(* CODESYS project PLS2 Trykkregulering 19.07.2021.export

Project tree, tasks and I/O mapping:
  application PLS2_Trykkregulering
    task PLC_Task (cyclic, interval 100 ms, priority 10, watchdog 90 ms x 1) calls PLC_PRG
    task TrendRecordingTask (cyclic, interval 100 ms, priority 15) calls VisuTrendStorageAccess.GlobalInstances.g_TrendRecordingManager.CyclicCall
    task VISU_TASK (cyclic, interval 100 ms, priority 15) calls VisuElems.Visu_Prg
    GlobalData/
      global variables HMI
      global variables IO
      global variables Local
      global variables SIM
      global variables STATUS
    program Alarms [ST]
    program Control [ST]
    program Initialize [ST]
    program Inputs [ST]
    program Outputs [ST]
    program PLC_PRG [ST]
    function RestartOpcUaMqttLinkOnDownload [ST]
    function RestartOpcUaMqttLinkOnOnlineChange [ST]
    program Simulation [ST]
    global variables PersistentVars
    visualisation Visualization
*)

// PLS2_Trykkregulering/PersistentVars
{attribute 'qualified_only'}
VAR_GLOBAL PERSISTENT RETAIN
	// Generated instance path of persistent variable
	HMI.AliveCounterPlc2Pv: AliveHmiPv;
	// Generated instance path of persistent variable
	HMI.DeliveryPump1Cmd: ControlAnalogHmiCmd;
	// Generated instance path of persistent variable
	HMI.DeliveryPump1Pv: ControlAnalogHmiPv;
	// Generated instance path of persistent variable
	HMI.DeliveryPump2Cmd: ControlAnalogHmiCmd;
	// Generated instance path of persistent variable
	HMI.DeliveryPump2Pv: ControlAnalogHmiPv;
	// Generated instance path of persistent variable
	HMI.DeliveryPump3Cmd: ControlAnalogHmiCmd;
	// Generated instance path of persistent variable
	HMI.DeliveryPump3Pv: ControlAnalogHmiPv;
	// Generated instance path of persistent variable
	HMI.DeliveryPumpPIDCmd: PIDHmiCmd;
	// Generated instance path of persistent variable
	HMI.DeliveryPumpPIDPv: PIDHmiPv;
	// Generated instance path of persistent variable
	HMI.DeliveryPumpWorkDistPv: WorkDistributorHmiPv;
	// Generated instance path of persistent variable
	HMI.TreatmentPressureCmd: SignalAnalogHmiCmd;
	// Generated instance path of persistent variable
	HMI.TreatmentPressurePv: SignalAnalogHmiPv;
	// Generated instance path of persistent variable
	HMI.ConsumerPressureCmd: SignalAnalogHmiCmd;
	// Generated instance path of persistent variable
	HMI.ConsumerPressurePv: SignalAnalogHmiPv;
END_VAR

// PLS2_Trykkregulering/GlobalData/HMI
{attribute 'qualified_only'}
VAR_GLOBAL PERSISTENT RETAIN
AliveCounterPlc2Pv:AliveHmiPv;

DeliveryPump1Cmd:ControlAnalogHmiCmd;
DeliveryPump1Pv:ControlAnalogHmiPv;
DeliveryPump2Cmd:ControlAnalogHmiCmd;
DeliveryPump2Pv:ControlAnalogHmiPv;
DeliveryPump3Cmd:ControlAnalogHmiCmd;
DeliveryPump3Pv:ControlAnalogHmiPv;
DeliveryPumpPIDCmd:PIDHmiCmd;
DeliveryPumpPIDPv:PIDHmiPv;
DeliveryPumpWorkDistPv:WorkDistributorHmiPv;
TreatmentPressureCmd:SignalAnalogHmiCmd;
TreatmentPressurePv:SignalAnalogHmiPv;
ConsumerPressureCmd:SignalAnalogHmiCmd;
ConsumerPressurePv:SignalAnalogHmiPv;
END_VAR

// PLS2_Trykkregulering/GlobalData/IO
{attribute 'qualified_only'}
VAR_GLOBAL
AI_DeliveryPump1SpeedPv:REAL;
AI_DeliveryPump2SpeedPv:Real;
AI_DeliveryPump3SpeedPv:Real;

AO_DeliveryPump1ControlValue:real;
AO_DeliveryPump2ControlValue:real;
AO_DeliveryPump3ControlValue:REAL;

AI_ConsumerPressurePv:REAL;
AI_TreatmentPressurePv:REAL;
END_VAR

// PLS2_Trykkregulering/GlobalData/Local
{attribute 'qualified_only'}
VAR_GLOBAL
DeliveryPump1:ControlAnalogFB;
DeliveryPump2:ControlAnalogFB;
DeliveryPump3:ControlAnalogFB;
DeliveryPumpPID:PIDFB;
DeliveryPumpWorkDist:WorkDistributorFB;
TreatmentPressure:SignalAnalogFB;
ConsumerPressure:SignalAnalogFB;
END_VAR

// PLS2_Trykkregulering/GlobalData/SIM
{attribute 'qualified_only'}
VAR_GLOBAL
	Disturbance:REAL;
	Process_y:REAL;
	Process:REAL;
	Ref:REAL;
	Output:REAL;
END_VAR

// PLS2_Trykkregulering/GlobalData/STATUS
{attribute 'qualified_only'}
VAR_GLOBAL
	OpcUaMqttLinkStatus: OpcUa_Mqtt_Status;
END_VAR

// PLS2_Trykkregulering/PLC_PRG
PROGRAM PLC_PRG
VAR
	_firstScan:BOOL := TRUE;
	_counter:INT;
	_lastRun:STRING;
END_VAR



// Signaling that the PLC is alive
Hmi.AliveCounterPlc2Pv._tagId := 'AliveCounterPlc2Pv';
Hmi.AliveCounterPlc2Pv._type := 'AliveHmi';
Hmi.AliveCounterPlc2Pv._owner := 'plc2';
HMI.AliveCounterPlc2Pv.CounterPv := HMI.AliveCounterPlc2Pv.CounterPv + 1;

_counter := STATUS.OpcUaMqttLinkStatus.AliveCounterPv;
_lastRun := STATUS.OpcUaMqttLinkStatus.LastRun;

IF _firstScan THEN
	Initialize();
END_IF
Inputs();
Alarms();
Control();
Outputs();
Simulation();





// Always last
_firstScan := FALSE;

END_PROGRAM

// PLS2_Trykkregulering/Initialize
PROGRAM Initialize
VAR
END_VAR



Hmi.DeliveryPumpPIDCmd.Tag := 'PID01';
Hmi.DeliveryPumpPIDCmd.Description := 'Regulator for controling pressure';
Hmi.DeliveryPumpPIDCmd.Auto := TRUE;
Hmi.DeliveryPumpPIDCmd.EnableK := TRUE;
Hmi.DeliveryPumpPIDCmd.EnableI := TRUE;
Hmi.DeliveryPumpPIDCmd.EnableD := TRUE;
Hmi.DeliveryPumpPIDCmd.K := 8.0;
Hmi.DeliveryPumpPIDCmd.Ti := 5.5;
Hmi.DeliveryPumpPIDCmd.Td := 0.5;
Hmi.DeliveryPumpPIDCmd.N := 10.0;
Hmi.DeliveryPumpPIDCmd.TrackingGain := 1.0;
Hmi.DeliveryPumpPIDCmd.u0 := 50.0;


HMI.DeliveryPump1Cmd.Tag := 'P01';
HMI.DeliveryPump1Cmd.Description := 'Delivery pump 1';
HMI.DeliveryPump1Cmd.Auto := TRUE;
HMI.DeliveryPump1Cmd.ManualControlValue_Cmd := 50.0;
HMI.DeliveryPump1Cmd.AlarmControlFailedLimit := 10.0;
HMI.DeliveryPump1Cmd.AlarmControlFailed.Description := 'Failed to control Delivery Pump 1';
HMI.DeliveryPump1Cmd.AlarmControlFailed.Delay.OnDelayLimit := 10.0;
HMI.DeliveryPump1Cmd.AlarmControlFailed.Delay.OffDelayLimit := 10.0;
HMI.DeliveryPump1Cmd.AlarmControlFailed.Acknowledged := TRUE;

HMI.DeliveryPump2Cmd.Tag := 'P02';
HMI.DeliveryPump2Cmd.Description := 'Delivery pump 2';
HMI.DeliveryPump2Cmd.Auto := TRUE;
HMI.DeliveryPump2Cmd.ManualControlValue_Cmd := 50.0;
HMI.DeliveryPump2Cmd.AlarmControlFailedLimit := 10.0;
HMI.DeliveryPump2Cmd.AlarmControlFailed.Description := 'Failed to control Delivery Pump 2';
HMI.DeliveryPump2Cmd.AlarmControlFailed.Delay.OnDelayLimit := 10.0;
HMI.DeliveryPump2Cmd.AlarmControlFailed.Delay.OffDelayLimit := 10.0;
HMI.DeliveryPump2Cmd.AlarmControlFailed.Acknowledged := TRUE;

HMI.DeliveryPump3Cmd.Tag := 'P03';
HMI.DeliveryPump3Cmd.Description := 'Delivery pump 2';
HMI.DeliveryPump3Cmd.Auto := TRUE;
HMI.DeliveryPump3Cmd.ManualControlValue_Cmd := 50.0;
HMI.DeliveryPump3Cmd.AlarmControlFailedLimit := 10.0;
HMI.DeliveryPump3Cmd.AlarmControlFailed.Description := 'Failed to control Delivery Pump 3';
HMI.DeliveryPump3Cmd.AlarmControlFailed.Delay.OnDelayLimit := 10.0;
HMI.DeliveryPump3Cmd.AlarmControlFailed.Delay.OffDelayLimit := 10.0;
HMI.DeliveryPump3Cmd.AlarmControlFailed.Acknowledged := TRUE;

Hmi.TreatmentPressureCmd.Tag := 'PT02';
Hmi.TreatmentPressureCmd.Description := 'Treatment pressure';
Hmi.TreatmentPressureCmd.AlarmHysteresis := 3.0;
Hmi.TreatmentPressureCmd.AlarmHighHighLimit := 90.0;
Hmi.TreatmentPressureCmd.AlarmHighLimit := 80.0;
Hmi.TreatmentPressureCmd.AlarmLowLowLimit := 10.0;
Hmi.TreatmentPressureCmd.AlarmLowLimit := 20.0;
Hmi.TreatmentPressureCmd.AlarmHigh.Description := 'High Treatment Pressure';
Hmi.TreatmentPressureCmd.AlarmHighHigh.Description := 'High high Treatment Pressure';
Hmi.TreatmentPressureCmd.AlarmLow.Description := 'Low Treatment Pressure';
Hmi.TreatmentPressureCmd.AlarmLowLow.Description := 'Low low Treatment Pressure';
Hmi.TreatmentPressureCmd.AlarmHigh.Delay.OnDelayLimit := 1.0;
Hmi.TreatmentPressureCmd.AlarmHigh.Delay.OffDelayLimit := 1.0;
Hmi.TreatmentPressureCmd.AlarmHighHigh.Delay.OnDelayLimit := 1.0;
Hmi.TreatmentPressureCmd.AlarmHighHigh.Delay.OffDelayLimit := 1.0;
Hmi.TreatmentPressureCmd.AlarmLow.Delay.OnDelayLimit := 1.0;
Hmi.TreatmentPressureCmd.AlarmLow.Delay.OffDelayLimit := 1.0;
Hmi.TreatmentPressureCmd.AlarmLowLow.Delay.OnDelayLimit := 1.0;
Hmi.TreatmentPressureCmd.AlarmLowLow.Delay.OffDelayLimit := 1.0;
Hmi.TreatmentPressureCmd.InputScaling.InputUnit := 'na';
Hmi.TreatmentPressureCmd.InputScaling.OutputUnit := 'bar';
Hmi.TreatmentPressureCmd.InputScaling.InputMax_Cmd := 100.0;
Hmi.TreatmentPressureCmd.InputScaling.InputMin_Cmd := 0.0;
Hmi.TreatmentPressureCmd.InputScaling.OutputMax_Cmd := 100.0;
Hmi.TreatmentPressureCmd.InputScaling.OutputMin_Cmd := 0.0;

Hmi.ConsumerPressureCmd.Tag := 'PT03';
Hmi.ConsumerPressureCmd.Description := 'Consumer pressure';
Hmi.ConsumerPressureCmd.AlarmHysteresis := 3.0;
Hmi.ConsumerPressureCmd.AlarmHighHighLimit := 90.0;
Hmi.ConsumerPressureCmd.AlarmHighLimit := 80.0;
Hmi.ConsumerPressureCmd.AlarmLowLowLimit := 10.0;
Hmi.ConsumerPressureCmd.AlarmLowLimit := 20.0;
Hmi.ConsumerPressureCmd.AlarmHigh.Description := 'High Consumer Pressure';
Hmi.ConsumerPressureCmd.AlarmHighHigh.Description := 'High high Consumer Pressure';
Hmi.ConsumerPressureCmd.AlarmLow.Description := 'Low Consumer Pressure';
Hmi.ConsumerPressureCmd.AlarmLowLow.Description := 'Low low Consumer Pressure';
Hmi.ConsumerPressureCmd.AlarmHigh.Delay.OnDelayLimit := 1.0;
Hmi.ConsumerPressureCmd.AlarmHigh.Delay.OffDelayLimit := 1.0;
Hmi.ConsumerPressureCmd.AlarmHighHigh.Delay.OnDelayLimit := 1.0;
Hmi.ConsumerPressureCmd.AlarmHighHigh.Delay.OffDelayLimit := 1.0;
Hmi.ConsumerPressureCmd.AlarmLow.Delay.OnDelayLimit := 1.0;
Hmi.ConsumerPressureCmd.AlarmLow.Delay.OffDelayLimit := 1.0;
Hmi.ConsumerPressureCmd.AlarmLowLow.Delay.OnDelayLimit := 1.0;
Hmi.ConsumerPressureCmd.AlarmLowLow.Delay.OffDelayLimit := 1.0;
Hmi.ConsumerPressureCmd.InputScaling.InputUnit := 'na';
Hmi.ConsumerPressureCmd.InputScaling.OutputUnit := 'bar';
Hmi.ConsumerPressureCmd.InputScaling.InputMax_Cmd := 100.0;
Hmi.ConsumerPressureCmd.InputScaling.InputMin_Cmd := 0.0;
Hmi.ConsumerPressureCmd.InputScaling.OutputMax_Cmd := 100.0;
Hmi.ConsumerPressureCmd.InputScaling.OutputMin_Cmd := 0.0;

END_PROGRAM

// PLS2_Trykkregulering/Control
PROGRAM Control
VAR
	
END_VAR



// Regulator block
Local.DeliveryPumpPID(_id := 'DeliveryPumpPID', _owner := 'plc2',
	InputReference := 6.0,
	ProcessMeasure := IO.AI_ConsumerPressurePv,
	Ts := 0.1,
	uMax := 100.0,
	uMin := 0.0,
	HmiCmd := Hmi.DeliveryPumpPIDCmd,
	HmiPv := Hmi.DeliveryPumpPIDPv);

// Work distribution
Local.DeliveryPumpWorkDist(_id := 'DeliveryPumpWorkDist', _owner := 'plc2',
	InputControlSignal := Local.DeliveryPumpPID.Output,
	Tag1 := Hmi.DeliveryPump1Cmd.Tag,
	Tag2 := Hmi.DeliveryPump2Cmd.Tag,
	Tag3 := Hmi.DeliveryPump3Cmd.Tag,
	InAuto1 := Hmi.DeliveryPump1Cmd.Auto,
	InAuto2 := Hmi.DeliveryPump2Cmd.Auto,
	InAuto3 := Hmi.DeliveryPump3Cmd.Auto,
	RunHours1 := Hmi.DeliveryPump1Pv.RunHours_Pv,
	RunHours2 := Hmi.DeliveryPump2Pv.RunHours_Pv,
	RunHours3 := Hmi.DeliveryPump3Pv.RunHours_Pv,
	ChangeInterval := 60.0,
	HmiPv := HMI.DeliveryPumpWorkDistPv);
	

// Pumps
Local.DeliveryPump1(_id := 'DeliveryPump1', _owner := 'plc2',
	HmiCmd := HMI.DeliveryPump1Cmd,
	HmiPv := HMI.DeliveryPump1Pv,
	Interlock := FALSE,
	Feedback := IO.AI_DeliveryPump1SpeedPv,
	ControlValueAuto_Cmd := Local.DeliveryPumpWorkDist.Out1);
	
Local.DeliveryPump2(_id := 'DeliveryPump2', _owner := 'plc2',
	HmiCmd := HMI.DeliveryPump2Cmd,
	HmiPv := HMI.DeliveryPump2Pv,
	Interlock := FALSE,
	Feedback := IO.AI_DeliveryPump2SpeedPv,
	ControlValueAuto_Cmd := Local.DeliveryPumpWorkDist.Out2);

Local.DeliveryPump3(_id := 'DeliveryPump3', _owner := 'plc2',
	HmiCmd := HMI.DeliveryPump3Cmd,
	HmiPv := HMI.DeliveryPump3Pv,
	Interlock := FALSE,
	Feedback := IO.AI_DeliveryPump3SpeedPv,
	ControlValueAuto_Cmd := Local.DeliveryPumpWorkDist.Out3);

END_PROGRAM

// PLS2_Trykkregulering/Inputs
PROGRAM Inputs
VAR
	
END_VAR


				
Local.TreatmentPressure(_id := 'TreatmentPressure', _owner := 'plc2',
				RawInput := IO.AI_TreatmentPressurePv,
				HmiCmd := HMI.TreatmentPressureCmd,
				HmiPv := HMI.TreatmentPressurePv);

Local.ConsumerPressure(_id := 'ConsumerPressure', _owner := 'plc2',
				RawInput := IO.AI_ConsumerPressurePv,
				HmiCmd := HMI.ConsumerPressureCmd,
				HmiPv := HMI.ConsumerPressurePv);

END_PROGRAM

// PLS2_Trykkregulering/Alarms
PROGRAM Alarms
VAR
END_VAR

END_PROGRAM

// PLS2_Trykkregulering/Outputs
PROGRAM Outputs
VAR
END_VAR



IO.AO_DeliveryPump1ControlValue := Local.DeliveryPump1.ControlValue;
IO.AO_DeliveryPump2ControlValue := Local.DeliveryPump2.ControlValue;
IO.AO_DeliveryPump3ControlValue := Local.DeliveryPump3.ControlValue;

END_PROGRAM

// PLS2_Trykkregulering/Simulation
PROGRAM Simulation
VAR
	_simDelay: ARRAY[0..20] OF REAL;
	_iprocess:INT := 13; // Endret fra 19 til 13. -Peder
	_idelay:INT := 0;
	pressureDisturbance: ARRAY[0..29] OF REAL := [ 0.9,
            0.9,
            0.85,
            0.85,
			0.8,
            0.8,
            0.75,
            0.75,
            0.7,
			0.75,
            0.75,
            0.8,
            0.8,
            0.85,
			0.85,
            0.9,
            0.9,
            0.95,
            0.95,
			1.0,
            1.0,
            1.05,
            1.05,
            1.1,
			1.1,
            1.05,
            1.05,
            1.0,
            0.95,
			0.9];
			timeNow: TIME;
			secondsNow:LWORD;
			fakeHour:LWORD;
			currentFakeHour:LWORD;
END_VAR

IO.AI_DeliveryPump1SpeedPv := IO.AO_DeliveryPump1ControlValue;
IO.AI_DeliveryPump2SpeedPv := IO.AO_DeliveryPump2ControlValue;
IO.AI_DeliveryPump3SpeedPv := IO.AO_DeliveryPump3ControlValue;

timeNow := TIME();
secondsNow := (TIME_TO_LWORD(timeNow)/1000) MOD 60;
fakeHour := secondsNow/2;
SIM.Disturbance := pressureDisturbance[fakeHour];
Sim.Output := Local.DeliveryPumpPID.Output;
Sim.Ref := HMI.DeliveryPumpPIDPv.Reference_Pv;

SIM.Process_y := process(u := _simDelay[_idelay MOD 19],
	Ts := 0.1, y := SIM.Process_Y, yMin := 0, yMax := 8.0, T :=5,  Kp := 1.0);
_idelay := _idelay + 1;

_simDelay[_iprocess MOD 19] :=((IO.AI_DeliveryPump1SpeedPv + IO.AI_DeliveryPump2SpeedPv + IO.AI_DeliveryPump3SpeedPv)/10);
_iprocess := _iprocess + 1;


SIM.Process:=SIM.Process_y-SIM.Disturbance;

IO.AI_ConsumerPressurePv := SIM.Process; 
IO.AI_TreatmentPressurePv := 5.0;

END_PROGRAM

// PLS2_Trykkregulering/RestartOpcUaMqttLinkOnDownload
FUNCTION RestartOpcUaMqttLinkOnDownload : DWORD
VAR_IN_OUT
	EventPrm: CmpApp.EVTPARAM_CmpApp;
END_VAR
VAR
END_VAR

(*
This function is called whan a download is about to happen. 
This will force the Opc Ua - MQTT link to restart.
The restart will take 10 seconds, allowing e!Cockpit to download and start before the link starts.
*)
Status.OpcUaMqttLinkStatus.Restart_Cmd := TRUE;

END_FUNCTION

// PLS2_Trykkregulering/RestartOpcUaMqttLinkOnOnlineChange
FUNCTION RestartOpcUaMqttLinkOnOnlineChange : DWORD
VAR_IN_OUT
	EventPrm: CmpApp.EVTPARAM_CmpApp;
END_VAR
VAR
END_VAR

(*
This function is called whan a online change is about to happen. 
This will force the Opc Ua - MQTT link to restart.
The restart will take 10 seconds, allowing e!Cockpit to download and start before the link starts.
*)
Status.OpcUaMqttLinkStatus.Restart_Cmd := TRUE;

END_FUNCTION

// PLS2_Trykkregulering/Visualization
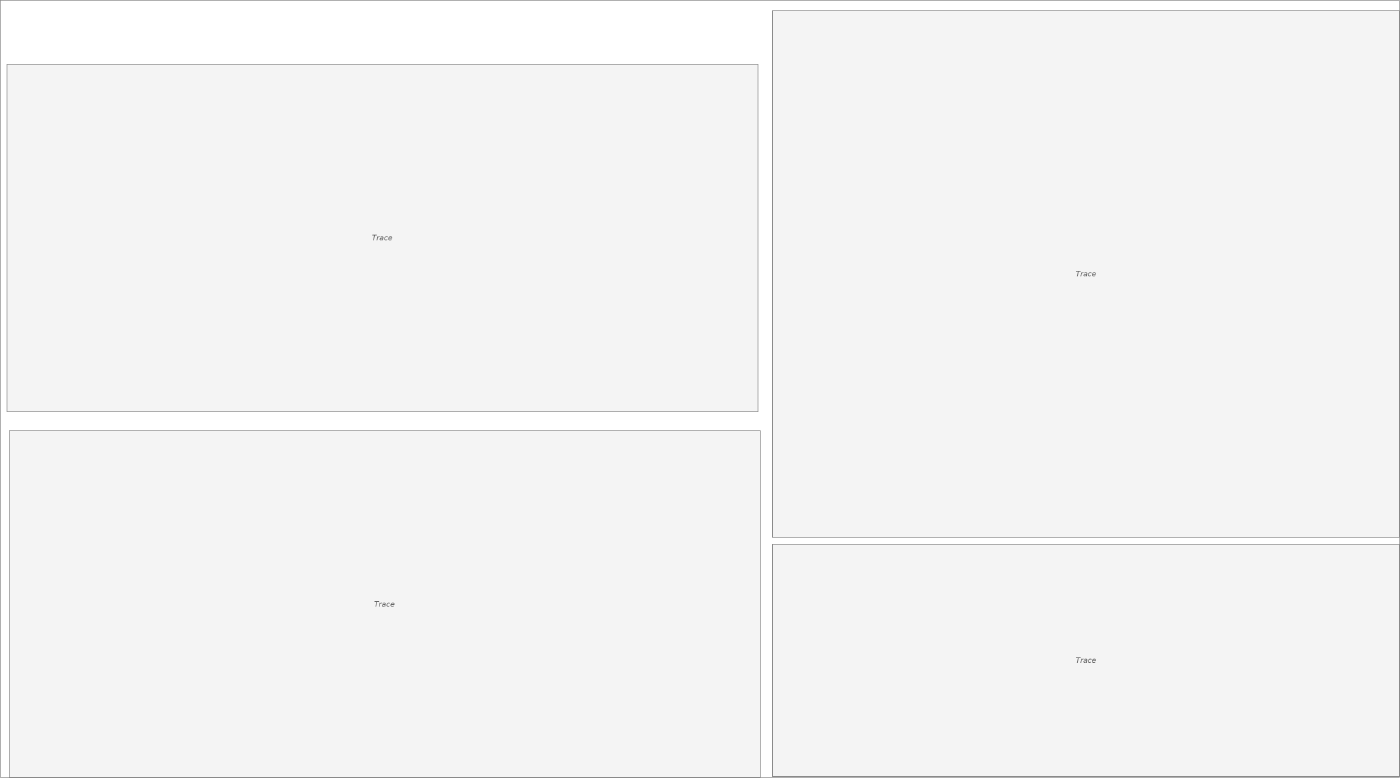
VISUALIZATION Visualization  // 1882x1047
    Trace (12,579 1010x468)
    Trace (1038,14 844x709)
    Trace (1038,732 844x313)
    Trace (9,86 1010x468)
END_VISUALIZATION
